{attribute addProperty BoxType "EPP4314-1002-0016"}
{attribute addProperty Id "Analog_outputAT %Q*INT162"}
{attribute addProperty CRC "4118783225"}
{attribute addProperty SizeInBites "16"}
{attribute addProperty SizeInBytes "2"}
TYPE AO_Standard_Channel_F57FA4F9 :
STRUCT
	{attribute addProperty Name "Analog_output"}
	Analog_output AT %Q* : INT;
END_STRUCT
END_TYPE

(* stored: Version 1.2.0.0, ProductVersion 3.1.4024.9
   DUT AO_Standard_Channel_F57FA4F9: Id {97b8ff57-93f1-4757-8e18-614298df0bb0} *)
